(* CoDeSys 2.3 export: EvtNull.EXP *)

(* POU core/evt/EvtNull, ST *)
FUNCTION EvtNull : BOOL
VAR_INPUT
END_VAR
VAR_IN_OUT
    Handle: LogBufferHandle;
END_VAR
VAR
    i: DINT;
    p1: POINTER TO BYTE;
END_VAR
i := GetNextWritePointer(4, Handle.BufferWritePointer, Handle.BufferReadPointer, Handle.BufferSize, Handle.BufferOverflow);
IF i >= 0 THEN

    p1 := Handle.BufferAddress + i;

    p1^ := START_FLAG;

    p1 := p1 + 1;
    p1^ := Handle.MagicByte;

    p1 := p1 + 1;
    p1^ := EVT_NULL;

    p1 := p1 + 1;
    p1^ := END_FLAG;

    Handle.BufferWritePointer := DWORD_TO_DINT(p1 - Handle.BufferAddress);

END_IF
END_FUNCTION
